TYPE ST_St040_HMI_OUT :
STRUCT
	//Pallet1,
	//Pallet2	: ST_Pallet;
END_STRUCT
END_TYPE

(* stored: Version 1.1.0.1
   DUT ST_St040_HMI_OUT: Id {2d3746a9-8257-4118-ba5e-c548aa441fb0} *)
